FUNCTION StartPump : BOOL
VAR_IN_OUT
	Pump	:	PumpType;
END_VAR
VAR
END_VAR

// start pump
Pump.RunState := Pumpstate.RUN;

END_FUNCTION

(* stored: Version 1.1.0.1, ProductVersion 3.1.4024.15
   POU StartPump: Id {61bd5ad0-4df3-4c26-ba25-4cae9e36c668}, SpecialFunc None *)
